FUNCTION_BLOCK ABSTRACT FB_Child2 EXTENDS FB_Parent

VAR
END_VAR

METHOD ABSTRACT Connect 
VAR_INPUT
END_VAR
END_METHOD

END_FUNCTION_BLOCK

(* stored: Version 1.1.0.1, ProductVersion 3.1.4024.16
   POU FB_Child2: Id {028d2de8-85d8-463e-96c5-d7f7a4125ac8}, SpecialFunc None
   Method Connect: Id {d232b42a-badc-44d7-98d4-7efe237174e2} *)
